TYPE ST_EventControl :
STRUCT

	ctrl		: ST_Event_Ctrl;
	stat		: ST_Event_Stat;

	Plc			: ST_PlcEvent;

END_STRUCT
END_TYPE

(* stored: Version 1.1.0.1, ProductVersion 3.1.4024.6
   DUT ST_EventControl: Id {1086bdd2-78dc-4bc8-8c4c-f6d47cf14e1b} *)
